TYPE ST_Tc3_DriveMotionControl :
STRUCT
	//Administrative/Axis Functions:
	Power 			: Tc3_DriveMotionControl.MC_Power;
	Reset           : Tc3_DriveMotionControl.MC_Reset;
	SetPosition     : Tc3_DriveMotionControl.MC_SetPosition;
	
	//Administrative/Touch Probe:
	AbortTrigger    : Tc3_DriveMotionControl.MC_AbortTrigger;
	TouchProbe      : Tc3_DriveMotionControl.MC_TouchProbe;
	
	//Motion/Homming:
	Home            : Tc3_DriveMotionControl.MC_Home;
	
	//Motion/Manual Motion:
	Jog             : Tc3_DriveMotionControl.MC_Jog;
	
	//Motion/Point to Point Motion:
	Halt            : Tc3_DriveMotionControl.MC_Halt;
	MoveAbsolute 	: Tc3_DriveMotionControl.MC_MoveAbsolute;
	MoveModulo      : Tc3_DriveMotionControl.MC_MoveModulo;
	MoveRelative 	: Tc3_DriveMotionControl.MC_MoveRelative;
	MoveVelocity    : Tc3_DriveMotionControl.MC_MoveVelocity;
	Stop            : Tc3_DriveMotionControl.MC_Stop;
END_STRUCT
END_TYPE

(* stored: Version 1.1.0.1, ProductVersion 3.1.4024.12
   DUT ST_Tc3_DriveMotionControl: Id {ccd99ec4-8598-47d9-b767-49a90359aee2} *)
